FUNCTION_BLOCK BfbCheck
  (* Standard: 61499-2 *)
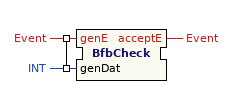
  EVENT_INPUT
    genE WITH genDat;
  END_EVENT
  EVENT_OUTPUT
    acceptE;
  END_EVENT
  VAR_INPUT
    genDat : INT := 1;
  END_VAR
  VAR
    comp : INT := 10;
    i : INT;
  END_VAR
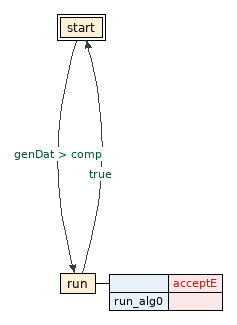
  EC_STATES
    start;
    run : -> acceptE, run_alg0;
  END_STATES
  EC_TRANSITIONS
    start TO run := genDat > comp;
    run TO start := true;
  END_TRANSITIONS
  ALGORITHM run_alg0 IN ST:
                if genDat > (comp + 5) then
                    for i := 0 to 10 by 2 do
                        comp := comp + genDat;
                    end_for;
                    printf("comp increased to:%d\n", comp);
                end_if;
  END_ALGORITHM
END_FUNCTION_BLOCK
